Yaskawa INFORM job: TWIN_FRONT_SEARCH_-90ST-2_5340.JBI

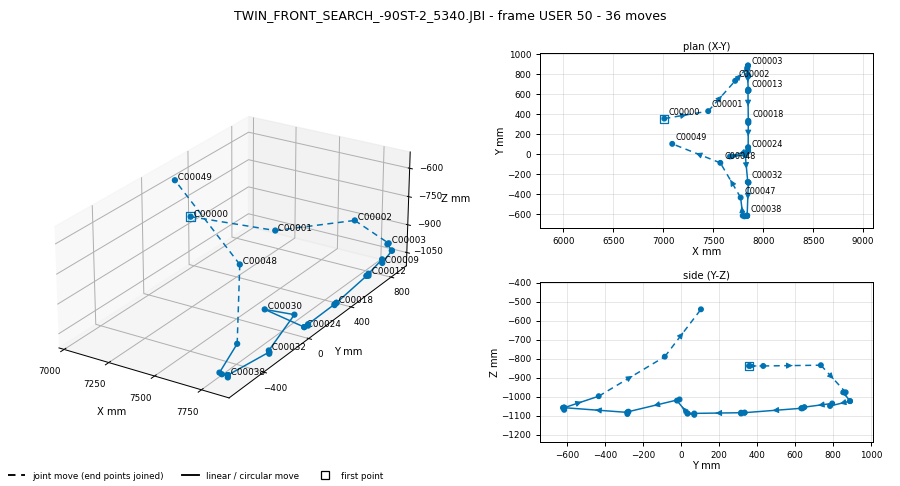
[picture p0: tool path of TWIN_FRONT_SEARCH_-90ST-2_5340.JBI in frame USER 50, 36 of 36 moves have a stored position in this frame; points joined in program order, loops and branches not executed]
/JOB
//NAME TWIN_FRONT_SEARCH_-90ST-2_5340
///FOLDERNAME 02-SKRZYNIE_JOBS
//POS
///NPOS 50,50,0,7,0,0
///USER 50
///TOOL 0
///POSTYPE USER
///RECTAN
///RCONF 1,0,0,0,0,0,0,0,0,0,0,0,0,0,0,0,0,0,0,0,0,0,0,0
C00000=7010.365,358.139,-838.637,56.3098,47.9541,-54.8379
C00001=7449.693,432.672,-838.681,56.3065,47.9522,-54.8413
C00002=7719.419,735.841,-834.672,56.3063,47.9500,-54.8422
C00003=7840.679,866.290,-977.211,38.5998,55.0414,-61.9603
C00004=7840.666,853.546,-977.206,32.5540,47.1319,-66.6775
C00005=7847.847,889.165,-1023.634,32.5585,47.1254,-66.6679
C00006=7847.854,889.161,-1041.100,32.5573,47.1259,-66.6703
C00007=7847.847,889.165,-1023.634,32.5585,47.1254,-66.6679
C00008=7848.341,903.073,-1029.326,32.5509,47.1214,-66.6762
C00009=7851.714,784.107,-1049.068,32.5585,47.1196,-66.6621
C00010=7870.522,784.116,-1049.072,32.5597,47.1194,-66.6606
C00011=7844.353,795.379,-1035.899,32.5565,47.1141,-66.6544
C00012=7849.782,649.232,-1055.038,32.5516,47.1138,-66.6549
C00013=7847.433,633.886,-1061.144,32.5484,47.1149,-66.6595
C00014=7847.456,633.875,-1074.972,32.5510,47.1138,-66.6562
C00015=7854.637,639.977,-1061.139,32.5477,47.1164,-66.6617
C00016=7869.302,637.485,-1061.149,32.5504,47.1135,-66.6540
C00017=7847.433,633.886,-1061.144,32.5484,47.1149,-66.6595
C00018=7850.734,334.573,-1084.328,31.8372,42.1263,-84.4315
///RCONF 0,0,0,0,0,0,0,0,0,0,0,0,0,0,0,0,0,0,0,0,0,0,0,0
C00019=7850.745,316.163,-1084.317,31.8376,42.1265,-84.4325
C00020=7850.741,316.160,-1094.362,31.8368,42.1262,-84.4329
C00021=7850.755,316.160,-1088.777,31.8376,42.1261,-84.4325
C00022=7865.576,316.144,-1088.767,31.8376,42.1256,-84.4340
///RCONF 1,0,0,0,0,0,0,0,0,0,0,0,0,0,0,0,0,0,0,0,0,0,0,0
C00023=7850.734,334.573,-1084.328,31.8372,42.1263,-84.4315
C00024=7849.357,34.560,-1088.545,31.8286,42.1352,-100.0040
///RCONF 0,0,0,0,0,0,0,0,0,0,0,0,0,0,0,0,0,0,0,0,0,0,0,0
C00025=7849.355,70.233,-1088.548,31.8281,42.1357,-100.0056
C00026=7849.345,70.212,-1100.998,31.8284,42.1333,-100.0035
C00027=7849.345,70.220,-1095.664,31.8295,42.1331,-100.0009
C00028=7865.259,70.222,-1095.685,31.8294,42.1306,-99.9970
///RCONF 1,0,0,0,0,0,0,0,0,0,0,0,0,0,0,0,0,0,0,0,0,0,0,0
C00029=7849.357,34.560,-1088.545,31.8286,42.1352,-100.0040
///RCONF 0,0,0,0,0,0,0,0,0,0,0,0,0,0,0,0,0,0,0,0,0,0,0,0
C00030=7667.857,-20.829,-1020.989,-0.6177,-11.3285,18.1841
///RCONF 1,0,0,0,0,0,0,0,0,0,0,0,0,0,0,0,0,0,0,0,0,0,0,0
C00031=7820.519,-7.380,-1014.685,-37.0724,25.7387,108.9100
C00032=7845.502,-275.775,-1078.939,-23.4713,44.5735,116.2747
C00033=7851.247,-281.568,-1082.953,-23.4687,44.5745,116.2764
C00034=7851.279,-281.525,-1093.483,-23.4710,44.5752,116.2796
C00035=7851.275,-281.534,-1091.324,-23.4693,44.5760,116.2816
C00036=7862.983,-281.554,-1091.347,-23.4675,44.5751,116.2800
C00037=7851.279,-281.526,-1082.832,-23.4696,44.5760,116.2817
C00038=7839.209,-614.059,-1058.152,-10.4658,52.1547,131.8418
C00039=7839.209,-614.059,-1058.152,-10.4658,52.1547,131.8418
C00040=7839.229,-614.033,-1075.081,-10.4663,52.1543,131.8452
///RCONF 0,0,0,0,0,0,0,0,0,0,0,0,0,0,0,0,0,0,0,0,0,0,0,0
C00041=7839.233,-614.011,-1069.388,-14.1441,54.0328,128.9016
C00042=7863.408,-614.027,-1069.387,-14.1410,54.0336,128.9042
///RCONF 1,0,0,0,0,0,0,0,0,0,0,0,0,0,0,0,0,0,0,0,0,0,0,0
C00043=7839.192,-614.061,-1058.166,-10.4648,52.1539,122.1660
C00044=7839.166,-656.145,-1058.183,-10.4641,52.1535,122.1647
///RCONF 0,0,0,0,0,0,0,0,0,0,0,0,0,0,0,0,0,0,0,0,0,0,0,0
C00045=7812.178,-620.370,-1058.486,-10.4558,52.1411,126.4774
C00046=7795.076,-613.348,-1058.098,-10.4617,52.1575,127.3673
///RCONF 1,0,0,0,0,0,0,0,0,0,0,0,0,0,0,0,0,0,0,0,0,0,0,0
C00047=7774.206,-432.297,-997.688,-17.4286,48.8596,123.7766
C00048=7570.999,-84.978,-789.821,-8.3295,54.7414,178.0447
C00049=7089.632,105.235,-540.772,34.6747,-14.1850,-36.1511
///RCONF 0,0,0,0,0,0,0,0,0,0,0,0,0,0,0,0,0,0,0,0,0,0,0,0
BC00000=5453.357
BC00001=5892.685
BC00002=6179.191
BC00003=6515.042
BC00004=6515.042
BC00005=6515.042
BC00006=6515.042
BC00007=6515.042
BC00008=6515.042
BC00009=6515.049
BC00010=6515.049
BC00011=6515.049
BC00012=6515.049
BC00013=6515.049
BC00014=6515.049
BC00015=6515.049
BC00016=6515.049
BC00017=6515.049
BC00018=6515.049
BC00019=6515.049
BC00020=6515.049
BC00021=6515.049
BC00022=6515.049
BC00023=6515.049
BC00024=6515.049
BC00025=6515.049
BC00026=6515.049
BC00027=6515.049
BC00028=6515.049
BC00029=6515.049
BC00030=6515.049
BC00031=6515.049
BC00032=6515.049
BC00033=6515.049
BC00034=6515.049
BC00035=6515.049
BC00036=6515.049
BC00037=6515.049
BC00038=6515.029
BC00039=6515.029
BC00040=6515.029
BC00041=6515.029
BC00042=6515.029
BC00043=6515.029
BC00044=6515.029
BC00045=6515.035
BC00046=6515.035
BC00047=6515.035
BC00048=6132.885
BC00049=5388.459
///POSTYPE BASE
P00006=-2.449,0.031,8.825,0.0000,0.0000,0.0000
///RCONF 1,0,0,0,0,0,0,0,0,0,0,0,0,0,0,0,0,0,0,0,0,0,0,0
P00500=2.332,-5.281,-1.258,0.0000,0.0000,0.0000
///RCONF 0,0,0,0,0,0,0,0,0,0,0,0,0,0,0,0,0,0,0,0,0,0,0,0
P00501=-2.026,0.009,3.534,0.0000,0.0000,0.0000
///RCONF 1,0,0,0,0,0,0,0,0,0,0,0,0,0,0,0,0,0,0,0,0,0,0,0
P00502=-2.023,0.001,1.732,0.0000,0.0000,0.0000
P00503=0.138,-0.044,1.539,0.0000,0.0000,0.0000
P00504=-0.309,-0.010,1.636,0.0000,0.0000,0.0000
P00505=0.999,-9.916,8.214,0.0000,0.0000,0.0000
//INST
///DATE 2024/10/28 16:27
///ATTR SC,RW,RJ
////FRAME USER 50
///GROUP1 RB1,BS1
NOP
MOVJ C00000 BC00000 VJ=30.00
MOVJ C00001 BC00001 VJ=50.00
MOVJ C00002 BC00002 VJ=50.00
MOVJ C00003 BC00003 VJ=30.00
'::::::::::::::::::::::::::::::::
'W21 P
'::::::::::::::::::::::::::::::::
MOVL C00004 BC00004 V=333.3
MOVL C00005 BC00005 V=166.7 PL=0
REFP 3 C00006 BC00006
CALL JOB:SEARCH-R1
SET P0500 P0006
SFTON P0500
MOVL C00007 BC00007 V=166.7 PL=0
REFP 3 C00008 BC00008
CALL JOB:SEARCH-R1
SET P0500 P0006
SFTON P0500
MOVL C00009 BC00009 V=166.7 PL=0
REFP 3 C00010 BC00010
CALL JOB:SEARCH-R1
SET P0500 P0006
SFTOF
MOVL C00011 BC00011 V=83.3
'::::::::::::::::::::::::::::::::
'W21 L
'::::::::::::::::::::::::::::::::
MOVL C00012 BC00012 V=250.0
MOVL C00013 BC00013 V=166.7 PL=0
REFP 3 C00014 BC00014
CALL JOB:SEARCH-R1
SET P0501 P0006
SFTON P0501
MOVL C00015 BC00015 V=166.7 PL=0
REFP 3 C00016 BC00016
CALL JOB:SEARCH-R1
SET P0501 P0006
SFTON P0501
MOVL C00017 BC00017 V=166.7 PL=0
SFTOF
'::::::::::::::::::::::::::::::::
'W20 P
'::::::::::::::::::::::::::::::::
MOVL C00018 BC00018 V=333.3
MOVL C00019 BC00019 V=166.7 PL=0
REFP 3 C00020 BC00020
CALL JOB:SEARCH-R1
SET P0502 P0006
SFTON P0502
MOVL C00021 BC00021 V=166.7 PL=0
REFP 3 C00022 BC00022
CALL JOB:SEARCH-R1
SET P0502 P0006
SFTON P0502
MOVL C00023 BC00023 V=166.7 PL=0
SFTOF
'::::::::::::::::::::::::::::::::
'W20 L
'::::::::::::::::::::::::::::::::
MOVL C00024 BC00024 V=250.0
MOVL C00025 BC00025 V=166.7 PL=0
REFP 3 C00026 BC00026
CALL JOB:SEARCH-R1
SET P0503 P0006
SFTON P0503
MOVL C00027 BC00027 V=66.7 PL=0
REFP 3 C00028 BC00028
CALL JOB:SEARCH-R1
SET P0503 P0006
SFTON P0503
MOVL C00029 BC00029 V=66.7 PL=0
SFTOF
'::::::::::::::::::::::::::::::::
'W22 P
'::::::::::::::::::::::::::::::::
MOVL C00030 BC00030 V=166.7
MOVL C00031 BC00031 V=166.7
MOVL C00032 BC00032 V=333.3
MOVL C00033 BC00033 V=166.7 PL=0
REFP 3 C00034 BC00034
CALL JOB:SEARCH-R1
SET P0504 P0006
SFTON P0504
MOVL C00035 BC00035 V=66.7 PL=0
REFP 3 C00036 BC00036
CALL JOB:SEARCH-R1
SET P0504 P0006
SFTON P0504
MOVL C00037 BC00037 V=66.7 PL=0
SFTOF
'::::::::::::::::::::::::::::::::
'W22 L
'::::::::::::::::::::::::::::::::
MOVL C00038 BC00038 V=333.3
MOVL C00039 BC00039 V=166.7 PL=0
REFP 3 C00040 BC00040
CALL JOB:SEARCH-R1
SET P0505 P0006
SFTON P0505
MOVL C00041 BC00041 V=166.7 PL=0
REFP 3 C00042 BC00042
CALL JOB:SEARCH-R1
SET P0505 P0006
SFTON P0505
MOVL C00043 BC00043 V=166.7 PL=0
REFP 3 C00044 BC00044
CALL JOB:SEARCH-R1
SET P0505 P0006
SFTOF
MOVL C00045 BC00045 V=83.3
MOVL C00046 BC00046 V=83.3
MOVL C00047 BC00047 V=250.0
MOVJ C00048 BC00048 VJ=40.00
MOVJ C00049 BC00049 VJ=80.00
END
